(* IEC 61131-3 sources: RL_MAR/experiments/comparison/llm4plc/results/gpt-4o-mini_20260506_100619/20260506_103703, 2 files *)

(* ---- generated_code_iteration_0.st ---- *)
ructured-text
FUNCTION_BLOCK DoughMixerControl
VAR_INPUT
    IngredientsDetected : BOOL; (* Input for detecting the presence of ingredients *)
END_VAR_INPUT

VAR_OUTPUT
    MixingInProgress : BOOL; (* Output for controlling the mixing process - on/off *)
END_VAR_OUTPUT

VAR
    MixingTimeElapsed : TIME; (* Timer to track the mixing time *)
    MixingTimeLimit : TIME := T#5S; (* Mixing time limit - 5 seconds *)
    prevIngredientsDetected : BOOL; (* To track the previous state of IngredientsDetected *)
END_VAR

(* Function Block Logic *)
IF IngredientsDetected AND NOT prevIngredientsDetected THEN
    MixingInProgress := TRUE; (* Start mixing *)
    MixingTimeElapsed := T#0S; (* Reset timer *)
ELSIF MixingInProgress THEN
    MixingTimeElapsed := MixingTimeElapsed + T#1S; (* Increment timer *)

    IF MixingTimeElapsed >= MixingTimeLimit OR NOT IngredientsDetected THEN
        MixingInProgress := FALSE; (* Stop mixing *)
    END_IF
END_IF

prevIngredientsDetected := IngredientsDetected; (* Update previous state *)
END_FUNCTION_BLOCK

(* ---- generated_code_iteration_1.st ---- *)
START_REASON
The errors in the original Structured Text (ST) code occurred due to incorrect usage of the variable declaration sections. Specifically, the output variable section was incorrectly closed with "END_VAR_OUTPUT" instead of the required "END_VAR". This caused the code to fail during the CODESYS compiler validation. Additionally, the overall structure of the function block needed to be maintained while ensuring proper syntax for variable declarations.
END_REASON

START_ST
FUNCTION_BLOCK DoughMixerControl
VAR_INPUT
    IngredientsDetected : BOOL; (* Input for detecting the presence of ingredients *)
END_VAR

VAR_OUTPUT
    MixingInProgress : BOOL; (* Output for controlling the mixing process - on/off *)
END_VAR

VAR
    MixingTimeElapsed : TIME; (* Timer to track the mixing time *)
    MixingTimeLimit : TIME := T#5S; (* Mixing time limit - 5 seconds *)
    prevIngredientsDetected : BOOL; (* To track the previous state of IngredientsDetected *)
END_VAR

(* Function Block Logic *)
IF IngredientsDetected AND NOT prevIngredientsDetected THEN
    MixingInProgress := TRUE; (* Start mixing *)
    MixingTimeElapsed := T#0S; (* Reset timer *)
ELSIF MixingInProgress THEN
    MixingTimeElapsed := MixingTimeElapsed + T#1S; (* Increment timer *)

    IF MixingTimeElapsed >= MixingTimeLimit OR NOT IngredientsDetected THEN
        MixingInProgress := FALSE; (* Stop mixing *)
    END_IF
END_IF

prevIngredientsDetected := IngredientsDetected; (* Update previous state *)
END_FUNCTION_BLOCK
END_ST
